
FUNCTION CB_sub_tod_t : TOD


TITLE = ' substracting a time of day from a duration '
VERSION : '1.0'
AUTHOR  : CB
NAME    : ad_tod_t
FAMILY  : TNI

VAR_INPUT
    IN0 : TOD;
    IN1 : TIME;
END_VAR

BEGIN
    CB_sub_tod_t := IN0 - IN1;
END_FUNCTION
